FUNCTION_BLOCK FB_ReactorLevelControl
VAR_INPUT
END_VAR
VAR_OUTPUT
	pressureControlOpen : BOOL; // Valve to control via pressure intervals
	timeControlOpen : BOOL; // Valve to control via on/off time intervals
END_VAR
VAR
	timeControlToggle: FB_ToggleHeartBeat;
	openInterval : INT;
	closeInterval : INT;
END_VAR

METHOD onOffTimeControl : BOOL
VAR_INPUT
	openIntervalSecs : INT; // Time for valve to stay open
	closeIntervalSecs : INT; // Time for valve to stay closed
END_VAR
openInterval := openIntervalSecs;
closeInterval := closeIntervalSecs ;
timeControlToggle(I_OpenInterValSecs := openInterval, I_CloseIntervalSecs := closeInterval, O_Update => timeControlOpen);
END_METHOD

METHOD pressureIntervalControl : BOOL
VAR_INPUT
	interval_1_condition: BOOL; // Condition for applying intervals marked with 1
	pressureUpperInterval_1 : INT;
	pressureLowerInterval_1 : INT;
	interval_2_condition: BOOL; // Condition for applying intervals marked with 2
	pressureUpperInterval_2 : INT;
	pressureLowerInterval_2 : INT;	
	interval_3_condition: BOOL; // Condition for applying intervals marked with 3
	pressureUpperInterval_3 : INT;
	pressureLowerInterval_3 : INT;	
	pressureValue : INT; // Pressure measurement
	pressureReference : INT; // Pressure reference (setpoint)
	valveOpenCondition : BOOL; // Condition for opening valve, must be filled for other factors to applu
	forceValveClosed : BOOL; // Condition for forcing valve closed independent of other factors
END_VAR

VAR
	pressureUpperInterval : INT;
	pressureLowerInterval: INT;
END_VAR
IF interval_1_condition THEN
	pressureUpperInterval := pressureUpperInterval_1;
	pressureLowerInterval := pressureLowerInterval_1;
ELSIF interval_2_condition THEN
	pressureUpperInterval := pressureUpperInterval_2;
	pressureLowerInterval := pressureLowerInterval_2;	
ELSIF interval_3_condition THEN
	pressureUpperInterval := pressureUpperInterval_3;
	pressureLowerInterval := pressureLowerInterval_3;		
END_IF

// Control valve when intervals are exceeded
IF (pressureValue >= pressureReference + pressureUpperInterval) AND valveOpenCondition THEN
	pressureControlOpen := TRUE;
ELSIF (pressureValue <= pressureReference - pressureLowerInterval) OR forceValveClosed THEN
	pressureControlOpen := FALSE;
END_IF
END_METHOD

END_FUNCTION_BLOCK

(* stored: Version 1.1.0.1, ProductVersion 3.1.4024.9
   POU FB_ReactorLevelControl: Id {ce7b3864-50f8-427a-82b3-cc6b587741b3}, SpecialFunc None
   Method onOffTimeControl: Id {32e4bde1-3926-4e59-a836-50da8d6efc09}
   Method pressureIntervalControl: Id {b27328fa-08a7-4d8f-a909-89cfa0a53987} *)
